// SIMATIC S7-200 project (STEP 7-Micro/WIN), CPU 221 REL 01.10

SYMBOL_TABLE USER1
MT               I0.0
MN               I0.1
ESTOP            I0.2
QT               Q0.0
QN               Q0.1
END_SYMBOL_TABLE

ORGANIZATION_BLOCK MAIN:OB1
TITLE=PROGRAM COMMENTS
BEGIN
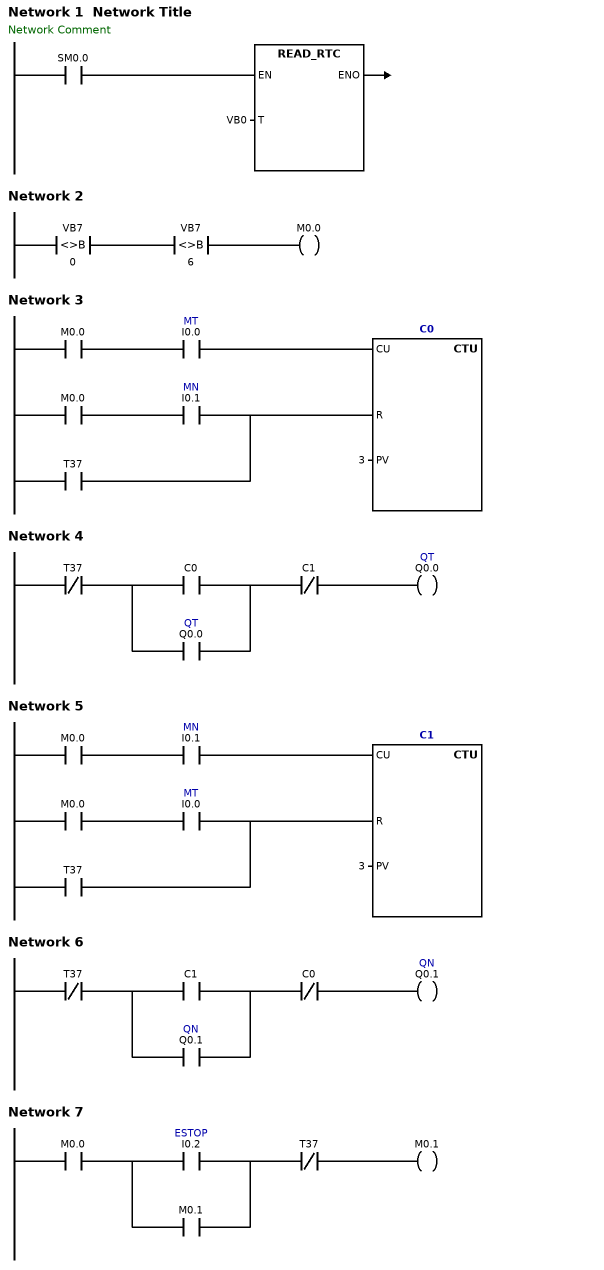
Network 1 // Network Title
// Network Comment
LD     SM0.0
TODR   VB0
Network 2
LDB<>  VB7, 0
AB<>   VB7, 6
=      M0.0
Network 3
LD     M0.0
A      MT:I0.0
LD     M0.0
A      MN:I0.1
O      T37
CTU    C0, 3
Network 4
LDN    T37
LD     C0
O      QT:Q0.0
ALD
AN     C1
=      QT:Q0.0
Network 5
LD     M0.0
A      MN:I0.1
LD     M0.0
A      MT:I0.0
O      T37
CTU    C1, 3
Network 6
LDN    T37
LD     C1
O      QN:Q0.1
ALD
AN     C0
=      QN:Q0.1
Network 7
LD     M0.0
LD     ESTOP:I0.2
O      M0.1
ALD
AN     T37
=      M0.1
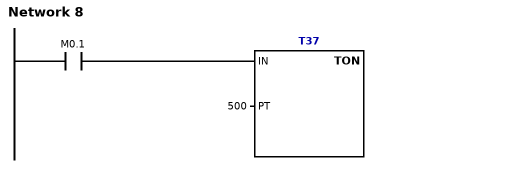
Network 8
LD     M0.1
TON    T37, 500
END_ORGANIZATION_BLOCK
